// TwinCAT 3 PLC project KbRail
// ProgramVersion: 3.1.4022.7
// libraries:
//   Tc2_MC2, * (Beckhoff Automation GmbH)
//   Tc2_Standard, * (Beckhoff Automation GmbH)
//   Tc2_System, * (Beckhoff Automation GmbH)
//   Tc3_Module, * (Beckhoff Automation GmbH)
//   VisuDialogs, * (System)
// project tree:
//   DUTs/ E_State.TcDUT, ST_AxisGroup.TcDUT
//   / GlobalTextList.TcGTLO, PlcTask.TcTTO, Visualization Manager.TcVMO (not stored)
//   POUs/ MAIN.TcPOU
//   VISUs/ Visualization.TcVIS
// real-time tasks:
//   TASK PlcTask: cycle T#10ms, priority 20, ADS port 350
// motion (NC):
//   TASK NC-Task 1 SAF: cycle T#2ms, priority 4, ADS port 501
//   TASK NC-Task 1 SVB: cycle T#10ms, priority 8, ADS port 511
//   AXIS Axis 1 (id 1)
//     Dynamic: AccelerationMaximum=0.6, DecelerationMaximum=0.6, Acceleration=0.59988, Deceleration=0.59988, Jerk=1.19952, DelayTime=0.008
//     Velo: Maximum=0.055
//     OtherSettings: AllowMotionCmdToSlave=true
//     encoder EncType=29
//       EncPara: ScaleFactorNumerator=1e-06, MaxCount=#xffffffff, EvaluationDirection=2
//         SoftEndMinControl: Enable=true, Range=1
//         Inc: RefSoftSyncMask=#x0000ffff
//     drive DrvType=24
//       DrvPara: Inverse=true
//         Analog: VeloReferenz=0.4, ScaleFactorActTorque=0.1
//         TimeComp: TaskDelayCycles=1
//     controller CtrType=1
//       CtrPara: PriorControlFactor=1
//         PosDiffControl: Range=0.2
//         Observer: BandWidth=20
// I/O:
//   DEVICE Device 1 (EtherCAT), AmsNetId 192.168.1.82.3.1
//     Term 12 (EK1100) [EK1100 EtherCAT Coupler (2A E-Bus)]
//       E1(EL7041) [EL7041 1Ch. Stepper motor output stage (50V, 5A)]
//       E2(EL5042) [EL5042 2Ch. BiSS-C Encoder]
//       E3(EL3202-0010)
//       Term 23 (EL9011) [EL9011 End Terminal]
// variable links:
//   NC-Task 1 SAF/Axes/Axis 1 <-> Device 1 (EtherCAT)/Term 12 (EK1100)/E1(EL7041)
//     Drive/Inputs/In/nState1 @bit 3 <-> STM Status/Status/Error
//     Drive/Inputs/In/nState1 @bit 5 <-> STM Status/Status/Moving negative
//     Drive/Inputs/In/nState1 @bit 4 <-> STM Status/Status/Moving positive
//     Drive/Inputs/In/nState1 @bit 1 <-> STM Status/Status/Ready
//     Drive/Inputs/In/nState1 <-> STM Status/Status/Ready to enable
//     Drive/Inputs/In/nState1 @bit 6 <-> STM Status/Status/Torque reduced
//     Drive/Inputs/In/nState1 @bit 2 <-> STM Status/Status/Warning
//     Drive/Inputs/In/nState2 @bit 5 <-> STM Status/Status/Sync error
//     Drive/Inputs/In/nState2 @bit 7 <-> STM Status/Status/TxPDO Toggle
//     Drive/Inputs/In/nState4 @bit 1 <-> WcState/InputToggle
//     Drive/Inputs/In/nState4 <-> WcState/WcState
//     Drive/Outputs/Out/nCtrl1 <-> STM Control/Control/Enable
//     Drive/Outputs/Out/nCtrl1 @bit 2 <-> STM Control/Control/Reduce torque
//     Drive/Outputs/Out/nCtrl1 @bit 1 <-> STM Control/Control/Reset
//     Drive/Outputs/Out/nDataOut2[0] <-> STM Velocity/Velocity
//   NC-Task 1 SAF/Axes/Axis 1 <-> Device 1 (EtherCAT)/Term 12 (EK1100)/E2(EL5042)
//     Enc/Inputs/In/nComState @bit 1 <-> WcState/InputToggle
//     Enc/Inputs/In/nComState <-> WcState/WcState
//     Enc/Inputs/In/nDataIn1 <-> FB Inputs Channel 1/Position
//     Enc/Inputs/In/nState1 @bit 12 <-> FB Inputs Channel 1/Status/Diag
//     Enc/Inputs/In/nState1 @bit 1 <-> FB Inputs Channel 1/Status/Error
//     Enc/Inputs/In/nState1 @bit 14 <-> FB Inputs Channel 1/Status/Input cycle counter
//     Enc/Inputs/In/nState1 @bit 2 <-> FB Inputs Channel 1/Status/Ready
//     Enc/Inputs/In/nState1 @bit 13 <-> FB Inputs Channel 1/Status/TxPDO State
//     Enc/Inputs/In/nState1 <-> FB Inputs Channel 1/Status/Warning
//   KbRail/KbRail Instance <-> Device 1 (EtherCAT)/Term 12 (EK1100)/E1(EL7041)
//     PlcTask Inputs/MAIN.M[1].bLimHigh <-> STM Status/Status/Digital input 1
//     PlcTask Inputs/MAIN.M[1].bLimLow <-> STM Status/Status/Digital input 2
//   KbRail/KbRail Instance <-> Device 1 (EtherCAT)/Term 12 (EK1100)/E3(EL3202-0010)
//     PlcTask Inputs/MAIN.RTD[1] <-> RTD Inputs Channel 1/Value
//     PlcTask Inputs/MAIN.RTD[2] <-> RTD Inputs Channel 2/Value
//   KbRail/KbRail Instance <-> NC-Task 1 SAF/Axes/Axis 1
//     PlcTask Inputs/MAIN.M[1].axisRef.NcToPlc <-> Outputs/ToPlc
//     PlcTask Outputs/MAIN.M[1].axisRef.PlcToNc <-> Inputs/FromPlc

CONFIGURATION KbRail
    RESOURCE PLC ON TwinCAT3
        TASK PlcTask(INTERVAL := T#10ms, PRIORITY := 20);
        PROGRAM MAIN WITH PlcTask : MAIN;
    END_RESOURCE
END_CONFIGURATION

// ---- DUTs/E_State.TcDUT
{attribute 'qualified_only'}
{attribute 'strict'}
TYPE E_State :
(
	idle,
	reset,
	moveAbs,
	moveRel
);
END_TYPE

// ---- DUTs/ST_AxisGroup.TcDUT
TYPE ST_AxisGroup :
STRUCT
	//basic built in functions
	mcPower		: MC_Power;
	mcReset		: MC_Reset;
	mcMoveAbs	: MC_MoveAbsolute;
	mcMoveRel	: MC_MoveRelative;
	mcHome		: MC_Home;
	mcStop		: MC_Stop;
	mcJog		: MC_Jog;
	
	//linkable variables
	axisRef				: AXIS_REF;;
	bLimHigh 	AT %I*	: BOOL;
	bLimLow 	AT %I*	: BOOL;

END_STRUCT
END_TYPE

// ---- POUs/MAIN.TcPOU
PROGRAM MAIN
VAR
	M			: ARRAY [1 .. 4] OF ST_AxisGroup;
	RTD AT %I*	: ARRAY [1 .. 4] OF INT;
	Temp1		: LREAL;
	Temp2		: LREAL;
	
	state		: E_State;
	fSpeed		: LREAL;
	fPosition	: LREAL;
	fPosRel		: LREAL;
	
END_VAR

(*update Axis_Ref status*)
M[1].axisRef.ReadStatus();
//M[2].axisRef.ReadStatus();
//M[3].axisRef.ReadStatus();
//M[4].axisRef.ReadStatus();

(*Enable motors*)
M[1].mcPower(Axis:=M[1].axisRef, Enable:=TRUE, Enable_Positive:=M[1].bLimHigh, Enable_Negative:=M[1].bLimLow);
//M[2].mcPower(Axis:=M[2].axisRef, Enable:=TRUE, Enable_Positive:=M[2].bLimHigh, Enable_Negative:=M[2].bLimLow);
//M[3].mcPower(Axis:=M[3].axisRef, Enable:=TRUE, Enable_Positive:=M[3].bLimHigh, Enable_Negative:=M[3].bLimLow);
//M[4].mcPower(Axis:=M[4].axisRef, Enable:=TRUE, Enable_Positive:=M[4].bLimHigh, Enable_Negative:=M[4].bLimLow);

Temp1:=INT_TO_LREAL(RTD[1])/100;
Temp2:=INT_TO_LREAL(RTD[2])/100;

IF (fSpeed>0.050) THEN
	fSpeed:=0.050;
ELSIF (fSpeed<0.00) THEN
	fSpeed:=0.00;
END_IF

CASE state OF
	E_State.idle:
		M[1].mcMoveAbs(Axis:=M[1].axisRef, Execute:=FALSE);
		M[1].mcMoveRel(Axis:=M[1].axisRef, Execute:=FALSE);
		M[1].mcReset(Axis:=M[1].axisRef, Execute:=FALSE);
	
	E_State.moveAbs:
		M[1].mcMoveRel(Axis:=M[1].axisRef, Execute:=FALSE);
		M[1].mcMoveAbs(Axis:=M[1].axisRef, Position:=fPosition, Velocity:=fSpeed, Execute:=TRUE);
		IF M[1].mcMoveAbs.Done THEN
			state:=E_State.idle;
		END_IF
	
	E_State.moveRel:
		M[1].mcMoveAbs(Axis:=M[1].axisRef, Execute:=FALSE);
		M[1].mcMoveRel(Axis:=M[1].axisRef, Distance:=fPosRel, Velocity:=fSpeed, Execute:=TRUE);
		IF M[1].mcMoveRel.Done THEN
			state:=E_State.idle;
		END_IF
		
	E_State.reset:
		M[1].mcReset(Axis:=M[1].axisRef, Execute:=TRUE);
		M[1].mcMoveAbs(Axis:=M[1].axisRef, Execute:=FALSE);
		M[1].mcMoveRel(Axis:=M[1].axisRef, Execute:=FALSE);
		IF M[1].mcReset.Done THEN
			state:=E_State.idle;
		END_IF
		
	ELSE
		M[1].mcReset(Axis:=M[1].axisRef, Execute:=TRUE);
		M[1].mcMoveAbs(Axis:=M[1].axisRef, Execute:=FALSE);
		M[1].mcMoveRel(Axis:=M[1].axisRef, Execute:=FALSE);
		IF M[1].mcReset.Done THEN
			state:=E_State.idle;
		END_IF
		
END_CASE

END_PROGRAM

// ---- GlobalTextList.TcGTLO
TEXTLIST GlobalTextList
  292 = '%7.1f'
  196 = '%7.3f'
  183 = '%7.4f'
  51 = 'adsf'
  3 = 'Current pos (mm): %7.4f'
  177 = 'Current Pos(mm): %7.1f'
  365 = 'Current Pos(mm): %7.4f'
  607 = 'Current Pos(mm):%7.1f'
  999 = 'Current Pos:%7.1f'
  6 = 'Current Temp (C): %5d'
  7 = 'Current Temp (C): %7.2f'
  8 = 'Current Temp (C): %7.3f'
  5 = 'Current Temp (C): %7.4f'
  84 = 'ERROR'
  733 = 'ERRORIn Motion'
  893 = 'Execute'
  444 = 'G'
  4 = 'GroupBox'
  910 = 'High Limit'
  502 = 'High Limit Activated'
  496 = 'High Limit Status'
  679 = 'In Motion'
  341 = 'IN MOTION'
  868 = 'Low Limit Status'
  571 = 'Move +100 um'
  529 = 'Move +50 um'
  472 = 'Move -100 um'
  19 = 'Move -50 um'
  853 = 'Move 50 um'
  393 = 'Move Absolute'
  327 = 'Move Relative'
  998 = 'Move to Position'
  986 = 'Move to Position:'
  936 = 'RESET/ABORT'
  140 = 'Set Position'
  1 = 'Set Position (mm)'
  594 = 'Set Position(mm)'
  835 = 'Set Speed'
  0 = 'Set Speed (mm)'
  2 = 'Set Speed (mm/s)'
  184 = 'Set Speed(mm/s)'
  66 = 'Status'
END_TEXTLIST

// ---- VISUs/Visualization.TcVIS
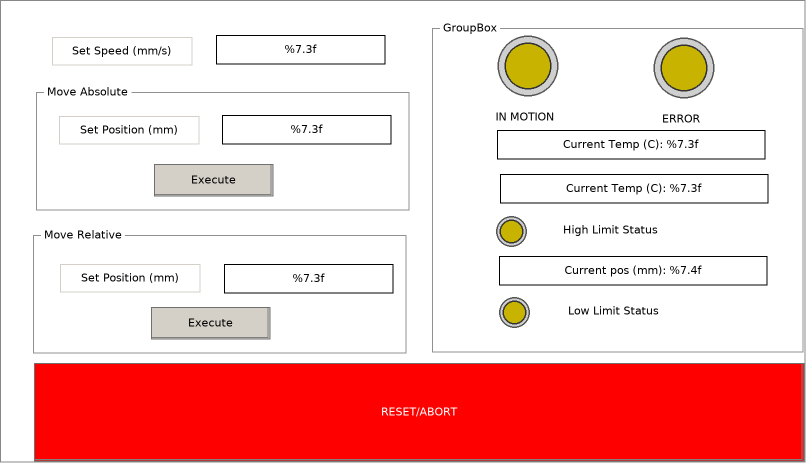
VISUALIZATION Visualization  // 806x463
    Rectangle (216,35 169x29), "%7.3f", text variable: MAIN.fSpeed
    Textfield (52,37 140x28), "Set Speed (mm/s)"
        OnMouseUp: write MAIN.fSpeed via Default, format %7.3f
    GroupBox (36,84 373x126), "Move Absolute"
        Button (118,80 119x32), "Execute"
            OnMouseUp: execute { MAIN.state:=E_State.moveAbs; }
        Rectangle (186,31 169x29), "%7.3f", text variable: MAIN.fPosition
        Textfield (23,32 140x28), "Set Position (mm)"
            OnMouseUp: write MAIN.fPosition via Default, format %7.3f
    GroupBox (33,227 373x126), "Move Relative"
        Button (118,80 119x32), "Execute"
            OnMouseUp: execute { MAIN.state:=E_State.moveRel; }
        Rectangle (191,37 169x29), "%7.3f", text variable: MAIN.fPosRel
        Textfield (27,37 140x28), "Set Position (mm)"
            OnMouseUp: write MAIN.fPosRel via Default, format %7.3f
    GroupBox (432,20 371x332), "GroupBox"
        Lamp1 (61,11 70x70), variable: MAIN.M[1].axisRef.Status.Moving, style: Lamp-Lamp1-Yellow
        Label (49,82 88x30), "IN MOTION"
        Lamp1 (217,13 70x70), variable: MAIN.M[1].mcMoveAbs.Error or MAIN.M[1].mcMoveRel.Error or MAIN.M[1].mcReset.Error, style: Lamp-Lamp1-Yellow
        Label (205,84 88x30), "ERROR"
        Lamp1 (62,192 35x39), variable: not(MAIN.M[1].bLimHigh), style: Lamp-Lamp1-Yellow
        Label (110,195 137x30), "High Limit Status"
        Lamp1 (65,273 35x39), variable: not(MAIN.M[1].bLimLow), style: Lamp-Lamp1-Yellow
        Label (113,276 137x30), "Low Limit Status"
        Rectangle (67,236 268x29), "Current pos (mm): %7.4f", text variable: MAIN.M[1].axisRef.NcToPlc.ActPos
        Rectangle (65,110 268x29), "Current Temp (C): %7.3f", text variable: MAIN.Temp1
        Rectangle (68,154 268x29), "Current Temp (C): %7.3f", text variable: MAIN.Temp2
    Button (34,363 770x98), "RESET/ABORT"
        OnMouseUp: execute { Main.state:=E_State.reset; }
END_VISUALIZATION
